// TwinCAT 3 PLC project TcoCognexVisionTests
// Title: TcoCognexVisionTests
// Company: Vortex.Library
// ProjectVersion: 0.6.0.913
// ProgramVersion: 3.1.4024.12
// libraries:
//   Tc2_Standard, * (Beckhoff Automation GmbH)
//   Tc2_System, * (Beckhoff Automation GmbH)
//   Tc3_Module, * (Beckhoff Automation GmbH)
//   TcoAbstractions, 0.6.0.913 (Vortex.Library)
//   TcoCognexVision, 0.6.0.913 (Vortex.Library)
//   TcoCore, 0.6.0.913 (Vortex.Library)
//   TcoInspectors, 0.6.0.913 (Vortex.Library)
//   TcoIo, 0.6.0.913 (Vortex.Library)
//   TcoUtilities, 0.6.0.913 (Vortex.Library)
// project tree:
//   DUTs/ DesignerResults.TcDUT, DesignerUserData.TcDUT
//   GVLs/ GVL.TcGVL
//   / PlcTask.TcTTO
//   POUs/ ITcoResultsData.TcIO, MAIN.TcPOU, myVeryFirstTcoContext.TcPOU, ProjectSpecificData.TcPOU
// (motion and I/O tree: see PLC project tcocognexvision)
// real-time tasks:
//   TASK PlcTask: cycle T#10ms, priority 20, ADS port 350
//   TASK PNIO: cycle T#8ms, priority 21, ADS port 351
// variable links:

CONFIGURATION TcoCognexVisionTests
    RESOURCE PLC ON TwinCAT3
        TASK PlcTask(INTERVAL := T#16ms, PRIORITY := 21);
        PROGRAM MAIN WITH PlcTask : MAIN;
    END_RESOURCE
END_CONFIGURATION

// ---- DUTs/DesignerResults.TcDUT
TYPE DesignerResults EXTENDS TcoCore.TcoStruct :
STRUCT
    {attribute addProperty Name "<#ResultBool#>"}
    ResultBool : BOOL;
    {attribute addProperty Name "<#ResultInt#>"}
    ResultInt : INT;
    {attribute addProperty Name "<#ResultString#>"}
    ResultString : STRING;
    {attribute addProperty Name "<#Data inspector#>"}
    DigitalInspector : TcoInspectors.TcoDigitalInspector(THISSTRUCT);
    {attribute addProperty Name "<#Data inspector#>"}
    DataInspector : TcoInspectors.TcoDataInspector(THISSTRUCT);
    {attribute addProperty Name "<#Analog inspector#>"}
    AnalogInspector : TcoInspectors.TcoAnalogueInspector(THISSTRUCT);
END_STRUCT
END_TYPE

// ---- DUTs/DesignerUserData.TcDUT
TYPE DesignerUserData EXTENDS TcoCore.TcoStruct :
STRUCT
    {attribute addProperty Name "<#ResultBool#>"}
    ResultBool : BOOL;
    {attribute addProperty Name "<#ResultInt#>"}
    ResultInt : INT;
    {attribute addProperty Name "<#ResultString#>"}
    ResultString : STRING;
END_STRUCT
END_TYPE

// ---- GVLs/GVL.TcGVL
{attribute 'qualified_only'}
VAR_GLOBAL
    myVeryFirstDatamanGVL : TcoCognexVision.TcoDatamanIO_v_5_x_x;
    myVeryFirstInsightGVL : TcoCognexVision.TcoInsightIO_v_5_x_x;
END_VAR

// ---- POUs/ITcoResultsData.TcIO
INTERFACE ITcoResultsData

END_INTERFACE

// ---- POUs/MAIN.TcPOU
PROGRAM MAIN
VAR
    myVeryFirstTcoContextInstance : myVeryFirstTcoContext;
END_VAR

myVeryFirstTcoContextInstance.Run();

END_PROGRAM

// ---- POUs/myVeryFirstTcoContext.TcPOU
FUNCTION_BLOCK myVeryFirstTcoContext EXTENDS TcoCore.TcoContext
VAR
    {attribute addProperty Name "<#My very first DATAMAN#>"}
    myVeryFirstDataman : TcoCognexVision.TcoDataman_v_5_x_x(THIS^);
    {attribute addProperty Name "<#My very first INSIGHT#>"}
    myVeryFirstInsight : TcoCognexVision.TcoInsight_v_5_x_x(THIS^);
    {attribute addProperty Name "<#Cognex Designer#>"}
    designer : TcoCognexVision.TcoDesigner_v_2_x_x(THIS^);
    {attribute addProperty Name "<#Project Specific Data#>"}
    _specificData : ProjectSpecificData(THIS^);
END_VAR

(*~
    <docu>
        <summary>
            Main method of the TcoContext. This is the entry point of any control logic that belongs to this context.
            The call of this method is ensured by calling the <c>InstanceName.Run()</c> method, and it must not be called explicitly.
            This method is abstract, and it must be overridden in derived block.
        </summary>
    </docu>
~*)
METHOD PROTECTED Main
VAR
END_VAR
myVeryFirstDataman(inoIoData := GVL.myVeryFirstDatamanGVL);
myVeryFirstDataman.Service();
myVeryFirstInsight.Config.UserDataSize := eTcoInsightUserDataSize_v_5_x_x.USER_DATA_128B;
myVeryFirstInsight.Config.ResultDataSize := eTcoInsightResultDataSize_v_5_x_x.RESULT_DATA_128B;
myVeryFirstInsight(inoIoData := GVL.myVeryFirstInsightGVL);
myVeryFirstInsight.Service();
myVeryFirstDataman.Read();
myVeryFirstDataman.GetResultAsString(0, myVeryFirstDataman.Status.SignalStatus.ResultLength);
designer(inoData := _specificData);
designer.Service();
END_METHOD

END_FUNCTION_BLOCK

// ---- POUs/ProjectSpecificData.TcPOU
FUNCTION_BLOCK ProjectSpecificData EXTENDS TcoCognexVision.TcoDesignerRootContainer
VAR_INPUT
END_VAR
VAR_OUTPUT
END_VAR
VAR
    {attribute wpf [Container(Layout.Stack,"PcToPlc")]}
    {attribute wpf [Group(Layout.GroupBox)]}
    {attribute addProperty Name "<#PcToPlc#>"}
    PcToPlc : DesignerResults;
    {attribute wpf [Container(Layout.Stack,"PlcToPc")]}
    {attribute wpf [Group(Layout.GroupBox)]}
    {attribute addProperty Name "<#PlcToPc#>"}
    PlcToPc : DesignerUserData;
END_VAR

PROPERTY PUBLIC Results : REFERENCE TO DesignerResults
GET
Results ref= PcToPlc;
END_GET
END_PROPERTY

PROPERTY PUBLIC UserData : REFERENCE TO DesignerUserData
GET
UserData ref= PlcToPc;
END_GET
END_PROPERTY

END_FUNCTION_BLOCK
